// TIA Portal V20 export
TYPE "MOTOR_LOCK_HMI_UDT"
   STRUCT
      State : DWord;   // Status Tec_Unit / State Tec_unit
      Plant_Identifier : WString[24];   // Betriebsmittel Kennzeichen / Plant identifier
      Move : Word;   // Schnittstelle Bewegungen / Interface Movement/Position
      Position : DWord;   // Schnittstelle Positionen 1-8 / Interface Position
      Alarm : Word;   // Störungen / Alarms
      State_Colour : SInt;   // Status Farbschema / State colour code
      HMI_Control_No : Int;   // HMI-Control Nummer / HMI-Control number
      OPModeArea { ExternalWritable := 'False'} : USInt;   // BA-Bereich / OPMode area
   END_STRUCT;
END_TYPE
